PROGRAM MAIN
VAR
myFB : FB_ClickLog;
minTime : TIME;
END_VAR

// NIET GETEST - CHATGPT GEMAAKT

myFB(); // Aanroepen van de FB in je programma
minTime := myFB.GetMinimumTime; // Haal de minimale tijd op

END_PROGRAM

(* stored: Version 1.1.0.1, ProductVersion 3.1.4024.12
   POU MAIN: Id {c58d287d-c62c-4c43-a4d1-fccc9fac33bc}, SpecialFunc None *)
